// SIMATIC S7-200 SMART project (STEP 7-Micro/WIN SMART), CPU ST20

SYMBOL_TABLE Table 1
Counter_1        C1
CON_Done         M0.0
CON_Busy         M0.1
CON_Error        M0.2
CON_Stat         MB1
SEND_Done        M2.0
SEND_Busy        M2.1
SEND_Error       M2.2
SEND_Stat        MB3
RECV_Done        M4.0
RECV_Busy        M4.1
RECV_Error       M4.2
RECV_Stat        MB5
RECV_Len         MW6
Counted          MW8
END_SYMBOL_TABLE

SYMBOL_TABLE System Symbols
Always_On        SM0.0    // Always ON
First_Scan_On    SM0.1    // ON for the first scan cycle only
END_SYMBOL_TABLE

ORGANIZATION_BLOCK MAIN:OB1
TITLE=Program Comments
BEGIN
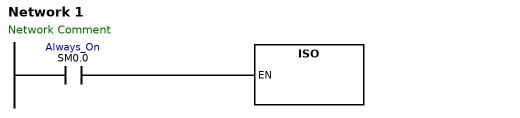
Network 1
// Network Comment
LD     Always_On:SM0.0
CALL   ISO:SBR10
END_ORGANIZATION_BLOCK

// SBR0: protected block, not included

SUBROUTINE_BLOCK ISO:SBR10
TITLE=Subroutine Comments
BEGIN
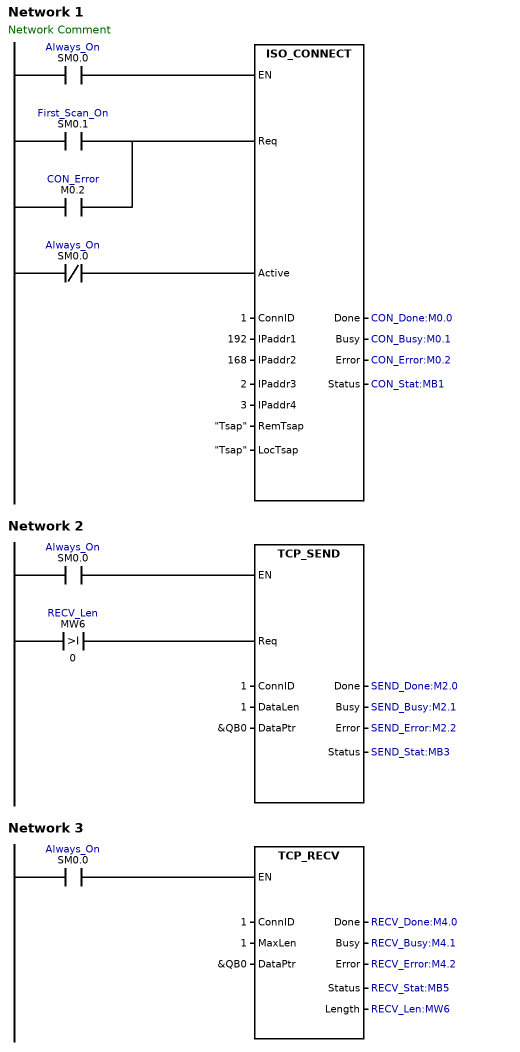
Network 1
// Network Comment
LD     Always_On:SM0.0
=      L60.0
LD     First_Scan_On:SM0.1
O      CON_Error:M0.2
=      L63.7
LDN    Always_On:SM0.0
=      L63.6
LD     L60.0
CALL   ISO_CONNECT:SBR11, L63.7, L63.6, 1, 192, 168, 2, 3, "Tsap", "Tsap", CON_Done:M0.0, CON_Busy:M0.1, CON_Error:M0.2, CON_Stat:MB1
Network 2
LD     Always_On:SM0.0
=      L60.0
LDW>   RECV_Len:MW6, 0
=      L63.7
LD     L60.0
CALL   TCP_SEND:SBR0, L63.7, 1, 1, &QB0, SEND_Done:M2.0, SEND_Busy:M2.1, SEND_Error:M2.2, SEND_Stat:MB3
Network 3
LD     Always_On:SM0.0
CALL   TCP_RECV:SBR13, 1, 1, &QB0, RECV_Done:M4.0, RECV_Busy:M4.1, RECV_Error:M4.2, RECV_Stat:MB5, RECV_Len:MW6
END_SUBROUTINE_BLOCK

// SBR11: protected block, not included

// SBR13: protected block, not included
